// TIA Portal V20 export
ORGANIZATION_BLOCK "DiagnosticErrorInterrupt"   // OB82, FBD, DiagnosticErrorInterrupt
{ S7_Optimized_Access := 'TRUE' }
// stored: SetENOAutomatically false
   VAR_INPUT
      IO_State : Word;   // IO state of the HW object
      LADDR : HW_ANY;   // Hardware identifier
      Channel : UInt;   // Channel number
      MultiError : Bool;   // =true if more than one error is present
   END_VAR
BEGIN

REGION Network 1: Submodul AI5/AQ2
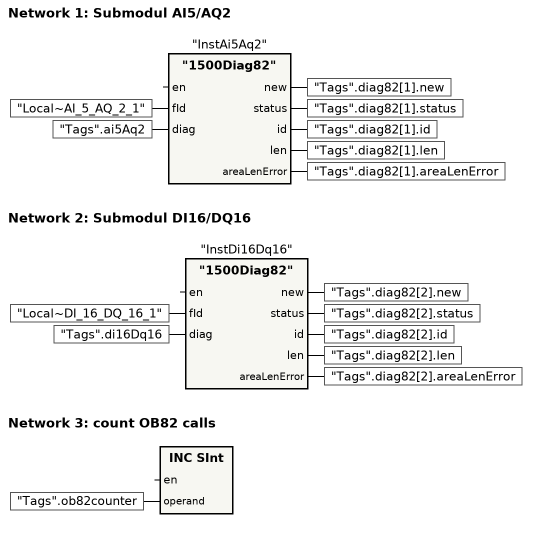
   "InstAi5Aq2"(fId := "Local~AI_5_AQ_2_1",   // "1500Diag82"
                diag := "Tags".ai5Aq2,
                new => "Tags".diag82[1].new,
                status => "Tags".diag82[1].status,
                id => "Tags".diag82[1].id,
                len => "Tags".diag82[1].len,
                areaLenError => "Tags".diag82[1].areaLenError);
END_REGION

REGION Network 2: Submodul DI16/DQ16
   "InstDi16Dq16"(fId := "Local~DI_16_DQ_16_1",   // "1500Diag82"
                  diag := "Tags".di16Dq16,
                  new => "Tags".diag82[2].new,
                  status => "Tags".diag82[2].status,
                  id => "Tags".diag82[2].id,
                  len => "Tags".diag82[2].len,
                  areaLenError => "Tags".diag82[2].areaLenError);
END_REGION

REGION Network 3: count OB82 calls
   "Tags".ob82counter := "Tags".ob82counter + 1;
END_REGION
END_ORGANIZATION_BLOCK
